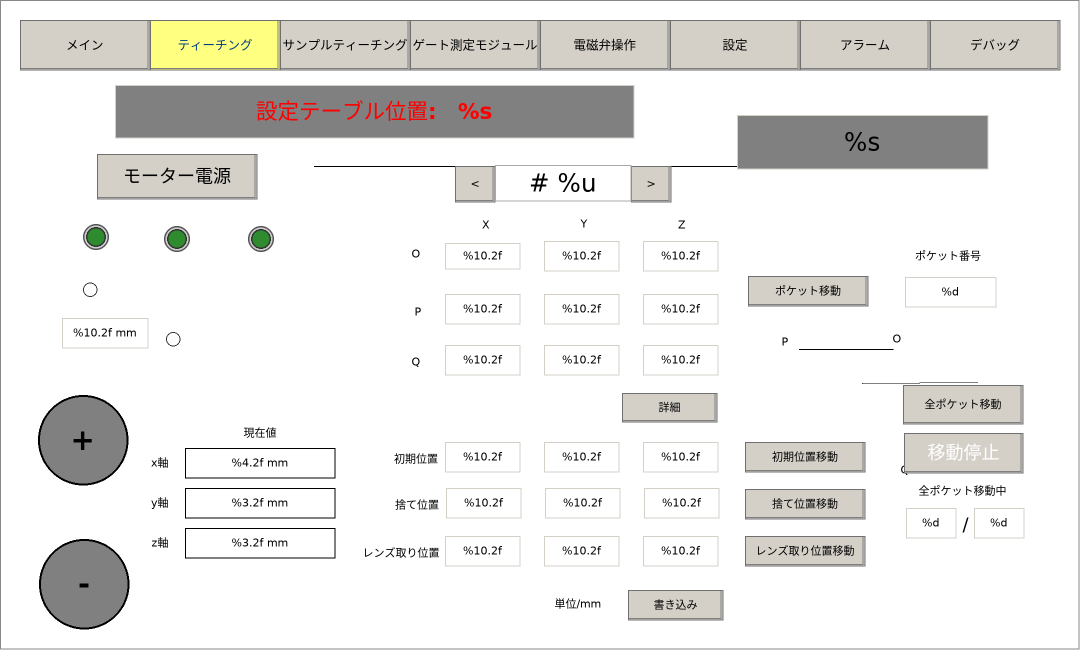
VISUALIZATION s_teaching1  // 1080x650
    Rectangle (0,0 1080x650)
    Lamp1 (246,224 30x30), variable: gvl_axis.fbi_mc_powerZ.Busy, style: Lamp-Lamp1-Green
    Lamp1 (162,224 30x30), variable: gvl_axis.fbi_mc_powerY.Busy, style: Lamp-Lamp1-Green
    Lamp1 (81,222 30x30), variable: gvl_axis.fbi_mc_powerX.Busy, style: Lamp-Lamp1-Green
    Textfield (445,243 75x26), "%10.2f", text variable: gvl_visu.var_in_palletizePos.Pos[1].x
        OnMouseClick: write gvl_visu.var_in_palletizePos.Pos[1].x via VisuDialogs.Numpad
    Textfield (445,294 75x30), "%10.2f", text variable: gvl_visu.var_in_palletizePos.Pos[2].x
        OnMouseClick: write gvl_visu.var_in_palletizePos.Pos[2].x via VisuDialogs.Numpad
    Textfield (445,345 75x30), "%10.2f", text variable: gvl_visu.var_in_palletizePos.Pos[3].x
        OnMouseClick: write gvl_visu.var_in_palletizePos.Pos[3].x via VisuDialogs.Numpad
    Label (391,347 50x30), "Q"
    Label (391,239 50x30), "O"
    Label (393,297 50x30), "P"
    Group (760,324 120x92)
        Line (39,25) (133,25)
        Line (102,59) (217,58)
        Label (112,0 50x30), "O"
        Label (0,3 50x30), "P"
        Label (120,131 50x30), "Q"
    Button (628,590 95x30), "書き込み"
        OnMouseClick: OpenDialog Dialog=d_saveBtn, OpenModal=True, OpenCentered=True
    Line (314,166) (799,166)
    Label (906,241 84x30), "ポケット番号", invisible if: gvl_visu.flg_All_PosPorket_Move
    Button (748,276 120x30), "ポケット移動", invisible if: gvl_axis.flg_motorReady = FALSE OR gvl_visu.flg_All_PosPorket_Move
        tap gvl_visu.flg_btn_PosPocket
    Textfield (62,318 86x30), "%10.2f mm", text variable: gvl_visu.var_in_inch
        OnMouseClick: write gvl_visu.var_in_inch via VisuDialogs.Numpad
    Textfield (544,241 75x30), "%10.2f", text variable: gvl_visu.var_in_palletizePos.Pos[1].y
        OnMouseClick: write gvl_visu.var_in_palletizePos.Pos[1].y via VisuDialogs.Numpad
    Textfield (643,241 75x30), "%10.2f", text variable: gvl_visu.var_in_palletizePos.Pos[1].z
        OnMouseClick: write gvl_visu.var_in_palletizePos.Pos[1].z via VisuDialogs.Numpad
    Textfield (544,294 75x30), "%10.2f", text variable: gvl_visu.var_in_palletizePos.Pos[2].y
        OnMouseClick: write gvl_visu.var_in_palletizePos.Pos[2].y via VisuDialogs.Numpad
    Textfield (643,294 75x30), "%10.2f", text variable: gvl_visu.var_in_palletizePos.Pos[2].z
        OnMouseClick: write gvl_visu.var_in_palletizePos.Pos[2].z via VisuDialogs.Numpad
    Textfield (544,345 75x30), "%10.2f", text variable: gvl_visu.var_in_palletizePos.Pos[3].y
        OnMouseClick: write gvl_visu.var_in_palletizePos.Pos[3].y via VisuDialogs.Numpad
    Textfield (643,345 75x30), "%10.2f", text variable: gvl_visu.var_in_palletizePos.Pos[3].z
        OnMouseClick: write gvl_visu.var_in_palletizePos.Pos[3].z via VisuDialogs.Numpad
    Label (461,210 50x30), "X"
    Label (559,209 50x30), "Y"
    Label (657,210 50x30), "Z"
    Textfield (445,442 75x30), "%10.2f", text variable: gvl_visu.var_in_initialPos.x
        OnMouseClick: write gvl_visu.var_in_initialPos.x via VisuDialogs.Numpad
    Label (391,444 50x30), "初期位置"
    Textfield (544,442 75x30), "%10.2f", text variable: gvl_visu.var_in_initialPos.y
        OnMouseClick: write gvl_visu.var_in_initialPos.y via VisuDialogs.Numpad
    Textfield (643,442 75x30), "%10.2f", text variable: gvl_visu.var_in_initialPos.z
        OnMouseClick: write gvl_visu.var_in_initialPos.z via VisuDialogs.Numpad
    Textfield (446,488 75x30), "%10.2f", text variable: gvl_visu.var_in_removePos.x
        OnMouseClick: write gvl_visu.var_in_removePos.x via VisuDialogs.Numpad
    Label (392,490 50x30), "捨て位置"
    Textfield (545,488 75x30), "%10.2f", text variable: gvl_visu.var_in_removePos.y
        OnMouseClick: write gvl_visu.var_in_removePos.y via VisuDialogs.Numpad
    Textfield (644,488 75x30), "%10.2f", text variable: gvl_visu.var_in_removePos.z
        OnMouseClick: write gvl_visu.var_in_removePos.z via VisuDialogs.Numpad
    Textfield (445,536 75x30), "%10.2f", text variable: gvl_visu.var_in_pickUpPos.x
        OnMouseClick: write gvl_visu.var_in_pickUpPos.x via VisuDialogs.Numpad
    Label (361,538 80x30), "レンズ取り位置"
    Textfield (544,536 75x30), "%10.2f", text variable: gvl_visu.var_in_pickUpPos.y
        OnMouseClick: write gvl_visu.var_in_pickUpPos.y via VisuDialogs.Numpad
    Textfield (643,536 75x30), "%10.2f", text variable: gvl_visu.var_in_pickUpPos.z
        OnMouseClick: write gvl_visu.var_in_pickUpPos.z via VisuDialogs.Numpad
    Button (745,442 120x30), "初期位置移動", invisible if: gvl_axis.flg_motorReady = FALSE
        tap gvl_visu.flg_btn_PosInit
    Button (745,489 120x30), "捨て位置移動", invisible if: gvl_axis.flg_motorReady = FALSE
        tap gvl_visu.flg_btn_PosRemove
    Button (745,536 120x30), "レンズ取り位置移動", invisible if: gvl_axis.flg_motorReady = FALSE
        tap gvl_visu.flg_btn_PosPickUP
    Label (135,448 50x30), "x軸"
    Label (135,488 50x30), "y軸"
    Label (135,528 50x30), "z軸"
    Rectangle (185,448 150x30), "%4.2f mm", text variable: gvl_axis.AxisX.NcToPlc.ActPos
    Rectangle (185,488 150x30), "%3.2f mm", text variable: gvl_axis.AxisY.NcToPlc.ActPos
    Rectangle (185,528 150x30), "%3.2f mm", text variable: gvl_axis.AxisZ.NcToPlc.ActPos
    RadioButton (81,270 249x39), variable: gvl_visu.var_jofAxis
    RadioButton (164,319 169x40), variable: gvl_visu.var_radio_jogMode
        Areas[0]: Text=インチ
        Areas[1]: Text=ジョグ
    Rectangle (737,115 251x54), "%s", text variable: gvl_param.var_productInfo[gvl_param.var_currentProductID].name
    Rectangle (115,85 519x53), "設定テーブル位置: %s", text variable: gvl_visu.var_currentTableMsg
    Ellipse (38,395 90x90), "+", invisible if: gvl_axis.flg_motorReady = FALSE
        OnMouseDown: execute { gvl_visu.flg_btn_moveDirct := eP_direction.positive; }
        OnMouseUp: execute { gvl_visu.flg_btn_moveDirct := eP_direction.keep; }
    Ellipse (39,539 90x90), "-", invisible if: gvl_axis.flg_motorReady = FALSE
        OnMouseDown: execute { gvl_visu.flg_btn_moveDirct := eP_direction.negative; }
        OnMouseUp: execute { gvl_visu.flg_btn_moveDirct := eP_direction.keep; }
    Textfield (905,277 91x30), "%d", text variable: gvl_visu.var_in_pocketNo, invisible if: gvl_visu.flg_All_PosPorket_Move
        OnMouseClick: write gvl_visu.var_in_pocketNo via VisuDialogs.Numpad
    Button (97,154 160x45), "モーター電源"
        toggle gvl_visu.flg_powerOn
    Button (622,393 95x29), "詳細"
        OnMouseClick: OpenDialog Dialog=d_teahingDetail, OpenModal=True, OpenCentered=True
    Button (20,20 130x50), "メイン"
        OnMouseClick: change screen: s_auto
    Button (150,20 130x50), "ティーチング"
        OnMouseClick: change screen: s_teaching1
    Button (670,20 130x50), "設定"
        OnMouseClick: change screen: s_setting
    Button (540,20 130x50), "電磁弁操作"
        OnMouseClick: change screen: s_manual
    Button (410,20 130x50), "ゲート測定モジュール"
        OnMouseClick: change screen: s_gm_teaching
    Button (800,20 130x50), "アラーム", colour toggle: gvl_io.flg_signalTowerRed
        OnMouseClick: change screen: s_alarm
    Button (280,20 130x50), "サンプルティーチング"
        OnMouseClick: change screen: s_sample
    Button (631,166 40x36), ">"
        OnMouseClick: execute {
            IF gvl_visu.var_in_cavNo < 8 THEN
            	gvl_visu.var_in_cavNo := gvl_visu.var_in_cavNo + 1;
            END_IF
        }
    Button (455,166 40x36), "<"
        OnMouseClick: execute {
            IF gvl_visu.var_in_cavNo > 1 THEN
            	gvl_visu.var_in_cavNo := gvl_visu.var_in_cavNo - 1;
            END_IF
        }
    Rectangle (495,165 136x36), "# %u", text variable: gvl_visu.var_in_cavNo
    Label (545,589 66x30), "単位/mm"
    Label (235,418 50x30), "現在値"
    Button (930,20 130x50), "デバッグ", colour toggle: gvl_io.flg_signalTowerRed
        OnMouseClick: change screen: s_debug
    Button (903,385 120x39), "全ポケット移動", invisible if: gvl_axis.flg_motorReady = FALSE OR gvl_visu.flg_All_PosPorket_Move
        tap gvl_visu.flg_btn_All_PosPocket
    Button (904,433 119x40), "移動停止", text variable: gvl_text.var_stopping, colour toggle: gvl_visu.flg_btn_autoModeStop, invisible if: NOT gvl_visu.flg_All_PosPorket_Move
        tap gvl_visu.flg_btn_autoModeStop
    Label (953,509 25x31), "/", invisible if: NOT gvl_visu.flg_All_PosPorket_Move
    Textfield (906,508 50x30), "%d", text variable: gvl_visu.var_in_pocketNo, invisible if: NOT gvl_visu.flg_All_PosPorket_Move
        OnMouseClick: write the text variable via VisuDialogs.Numpad
    Textfield (974,508 50x30), "%d", text variable: gvl_param.var_productInfo[gvl_param.var_currentProductID].pocketSumQty, invisible if: NOT gvl_visu.flg_All_PosPorket_Move
        OnMouseClick: write the text variable via VisuDialogs.Numpad
    Label (908,476 109x30), "全ポケット移動中", invisible if: NOT gvl_visu.flg_All_PosPorket_Move
END_VISUALIZATION

(* stored: Version 1.1.0.1, ProductVersion 3.1.4024.11
   Visu s_teaching1: Id {2bd95129-bb7d-4229-b553-b2023c6afe67} *)
